{attribute 'qualified_only'}
// Cooked IO aliases. Bound to the raw GVL_IO.dIn[i]/dOut[i] hardware arrays
// in MAIN's read-inputs / write-outputs bookends. No AT %*: these are plain
// BOOLs the FBs consume — the actual hardware wiring lives in GVL_IO.
//
// Tag convention: <Device>Sol<N>  = single EXTEND coil (SOL-Spring).
// The mechanical spring returns the actuator when the coil is de-energised,
// so no per-actuator Retract alias exists. DI still has a Retracted sensor.
//
//   SepSolN : Pin separator N   (DI 1..6, DO 1..3)
//   PushSolN: Pin push N        (DI 7..12, DO 4..6)
//   GripSolL / GripSolR: side grip pistons that clamp the robot-placed plate
//                       (DI 14..17, DO 8..9)
//   PlateSenL / PlateSenR: plate-presence sensors gating cycle start
//                         (DI 18..19)
//
// DO layout:
//   dOut[1..3] = SepSolN Extend
//   dOut[4..6] = PushSolN Extend
//   dOut[7]    = Robot bAssemblyRunning
//   dOut[8..9] = GripSolL/R Extend
//   dOut[10..16] = free
VAR_GLOBAL
    // SepSol1 (Pin separator 1) — DI 1..2, DO 1
    bSensorSepRetracted1  : BOOL;
    bSensorSepExtended1   : BOOL;
    bValveSepExtend1      : BOOL;

    // SepSol2 (Pin separator 2) — DI 3..4, DO 2
    bSensorSepRetracted2  : BOOL;
    bSensorSepExtended2   : BOOL;
    bValveSepExtend2      : BOOL;

    // SepSol3 (Pin separator 3) — DI 5..6, DO 3
    bSensorSepRetracted3  : BOOL;
    bSensorSepExtended3   : BOOL;
    bValveSepExtend3      : BOOL;

    // PushSol1 (Pin push 1) — DI 7..8, DO 4
    bSensorPushRetracted1 : BOOL;
    bSensorPushExtended1  : BOOL;
    bValvePushExtend1     : BOOL;

    // PushSol2 (Pin push 2) — DI 9..10, DO 5
    bSensorPushRetracted2 : BOOL;
    bSensorPushExtended2  : BOOL;
    bValvePushExtend2     : BOOL;

    // PushSol3 (Pin push 3) — DI 11..12, DO 6
    bSensorPushRetracted3 : BOOL;
    bSensorPushExtended3  : BOOL;
    bValvePushExtend3     : BOOL;

    // GripSolL (side grip, left) — DI 14..15, DO 8
    bSensorGripRetractedL : BOOL;
    bSensorGripExtendedL  : BOOL;
    bValveGripExtendL     : BOOL;

    // GripSolR (side grip, right) — DI 16..17, DO 9
    bSensorGripRetractedR : BOOL;
    bSensorGripExtendedR  : BOOL;
    bValveGripExtendR     : BOOL;

    // Plate-presence sensors — DI 18..19 (input only; no coil)
    bPlateSenL : BOOL;
    bPlateSenR : BOOL;
END_VAR

(* stored: Version 1.1.0.1, ProductVersion 3.1.4026.18
   GVL GVL_App: Id {f7ee3213-c403-4290-aff3-682ca99b3920} *)
